// TIA Portal V20 export
TYPE "LER_typeSleepMode"
// stored: Access Published
   STRUCT
      Normal : Bool;
      Idle : Bool;
      SleepTransition : Bool;
      Sleep : Bool;
      DeepSleepTransition : Bool;
      DeepSleep : Bool;
      WakeupRecovery : Bool;
   END_STRUCT;
END_TYPE
